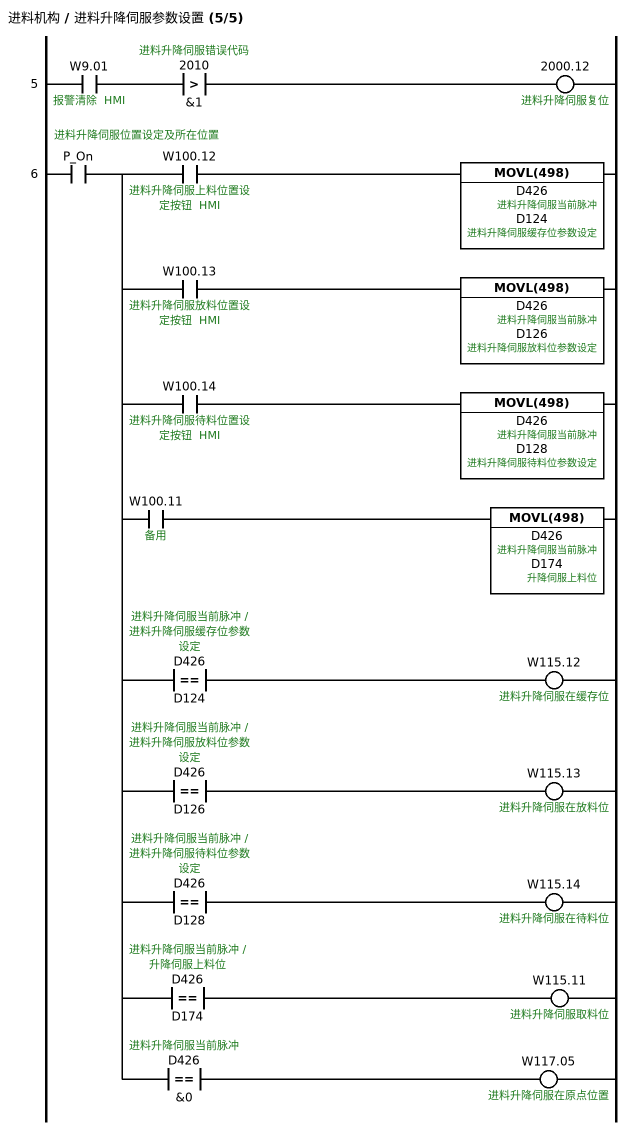
; [picture p144: 进料机构 / 进料升降伺服参数设置, rungs 5-6]
; rung 5
LD W9.01  ; 报警清除  HMI
AND>(320) 2010 &1  ; 进料升降伺服错误代码
OUT 2000.12  ; 进料升降伺服复位
; rung 6: 进料升降伺服位置设定及所在位置
LD P_On
OUT TR0
AND W100.12  ; 进料升降伺服上料位置设定按钮  HMI
MOVL(498) D426 D124  ; 进料升降伺服当前脉冲, 进料升降伺服缓存位参数设定
LD TR0
AND W100.13  ; 进料升降伺服放料位置设定按钮  HMI
MOVL(498) D426 D126  ; 进料升降伺服当前脉冲, 进料升降伺服放料位参数设定
LD TR0
AND W100.14  ; 进料升降伺服待料位置设定按钮  HMI
MOVL(498) D426 D128  ; 进料升降伺服当前脉冲, 进料升降伺服待料位参数设定
LD TR0
AND W100.11  ; 备用
MOVL(498) D426 D174  ; 进料升降伺服当前脉冲, 升降伺服上料位
LD TR0
AND=(300) D426 D124  ; 进料升降伺服当前脉冲, 进料升降伺服缓存位参数设定
OUT W115.12  ; 进料升降伺服在缓存位
LD TR0
AND=(300) D426 D126  ; 进料升降伺服当前脉冲, 进料升降伺服放料位参数设定
OUT W115.13  ; 进料升降伺服在放料位
LD TR0
AND=(300) D426 D128  ; 进料升降伺服当前脉冲, 进料升降伺服待料位参数设定
OUT W115.14  ; 进料升降伺服在待料位
LD TR0
AND=(300) D426 D174  ; 进料升降伺服当前脉冲, 升降伺服上料位
OUT W115.11  ; 进料升降伺服取料位
LD TR0
AND=(300) D426 &0  ; 进料升降伺服当前脉冲
OUT W117.05  ; 进料升降伺服在原点位置

### Section 进料旋转伺服参数设置

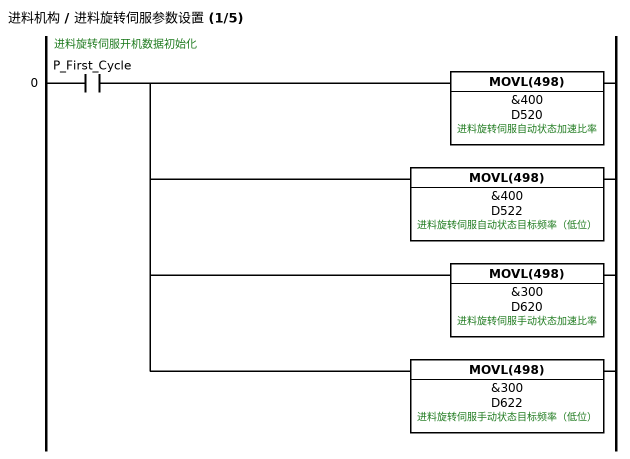
; rung 0: 进料旋转伺服开机数据初始化
LD P_First_Cycle
MOVL(498) &400 D520  ; 进料旋转伺服自动状态加速比率
MOVL(498) &400 D522  ; 进料旋转伺服自动状态目标频率（低位）
MOVL(498) &300 D620  ; 进料旋转伺服手动状态加速比率
MOVL(498) &300 D622  ; 进料旋转伺服手动状态目标频率（低位）

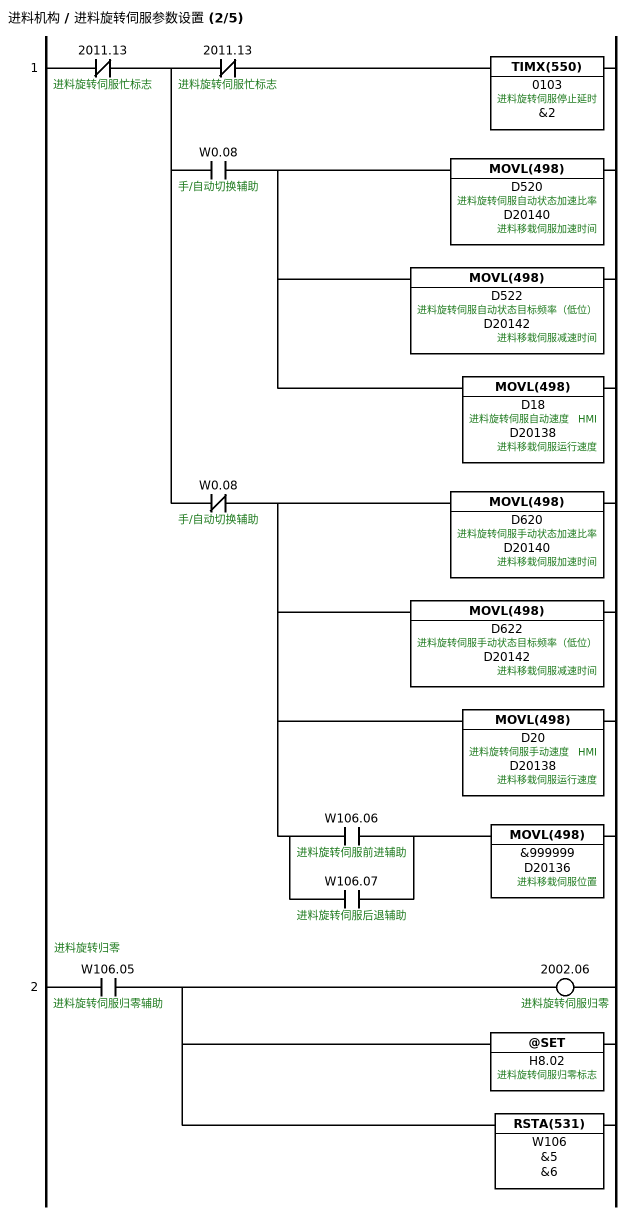
; rung 1
LDNOT 2011.13  ; 进料旋转伺服忙标志
OUT TR0
ANDNOT 2011.13  ; 进料旋转伺服忙标志
TIMX(550) 0103 &2  ; 进料旋转伺服停止延时
LD TR0
AND W0.08  ; 手/自动切换辅助
MOVL(498) D520 D20140  ; 进料旋转伺服自动状态加速比率, 进料移栽伺服加速时间
MOVL(498) D522 D20142  ; 进料旋转伺服自动状态目标频率（低位）, 进料移栽伺服减速时间
MOVL(498) D18 D20138  ; 进料旋转伺服自动速度   HMI, 进料移栽伺服运行速度
LD TR0
ANDNOT W0.08  ; 手/自动切换辅助
MOVL(498) D620 D20140  ; 进料旋转伺服手动状态加速比率, 进料移栽伺服加速时间
MOVL(498) D622 D20142  ; 进料旋转伺服手动状态目标频率（低位）, 进料移栽伺服减速时间
MOVL(498) D20 D20138  ; 进料旋转伺服手动速度   HMI, 进料移栽伺服运行速度
LD W106.06  ; 进料旋转伺服前进辅助
OR W106.07  ; 进料旋转伺服后退辅助
ANDLD
MOVL(498) &999999 D20136  ; 进料移栽伺服位置
; rung 2: 进料旋转归零
LD W106.05  ; 进料旋转伺服归零辅助
OUT 2002.06  ; 进料旋转伺服归零
@SET H8.02  ; 进料旋转伺服归零标志
RSTA(531) W106 &5 &6

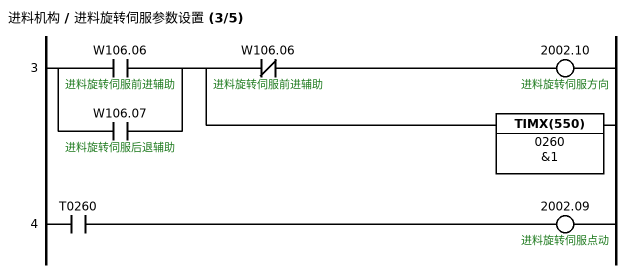
; rung 3
LD W106.06  ; 进料旋转伺服前进辅助
OR W106.07  ; 进料旋转伺服后退辅助
OUT TR0
ANDNOT W106.06  ; 进料旋转伺服前进辅助
OUT 2002.10  ; 进料旋转伺服方向
LD TR0
TIMX(550) 0260 &1
; rung 4
LD T0260
OUT 2002.09  ; 进料旋转伺服点动

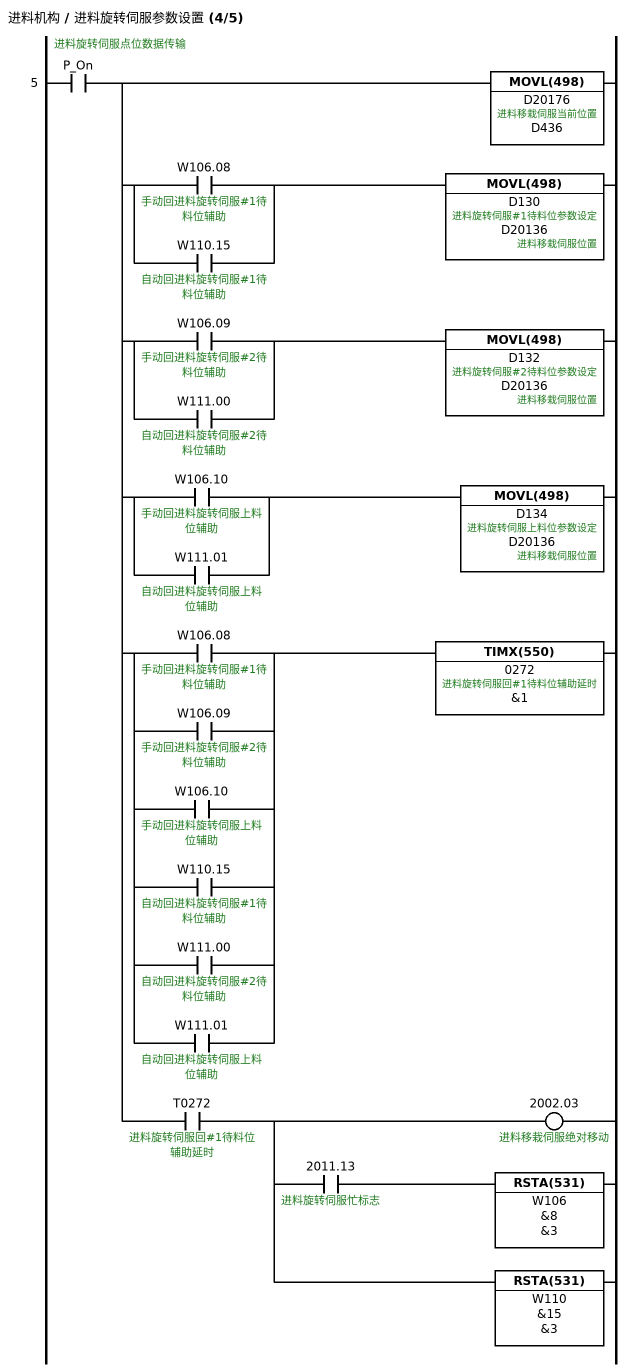
; rung 5: 进料旋转伺服点位数据传输
LD P_On
OUT TR0
MOVL(498) D20176 D436  ; 进料移栽伺服当前位置
LD W106.08  ; 手动回进料旋转伺服#1待料位辅助
OR W110.15  ; 自动回进料旋转伺服#1待料位辅助
ANDLD
MOVL(498) D130 D20136  ; 进料旋转伺服#1待料位参数设定, 进料移栽伺服位置
LD TR0
LD W106.09  ; 手动回进料旋转伺服#2待料位辅助
OR W111.00  ; 自动回进料旋转伺服#2待料位辅助
ANDLD
MOVL(498) D132 D20136  ; 进料旋转伺服#2待料位参数设定, 进料移栽伺服位置
LD TR0
LD W106.10  ; 手动回进料旋转伺服上料位辅助
OR W111.01  ; 自动回进料旋转伺服上料位辅助
ANDLD
MOVL(498) D134 D20136  ; 进料旋转伺服上料位参数设定, 进料移栽伺服位置
LD TR0
LD W106.08  ; 手动回进料旋转伺服#1待料位辅助
OR W106.09  ; 手动回进料旋转伺服#2待料位辅助
OR W106.10  ; 手动回进料旋转伺服上料位辅助
OR W110.15  ; 自动回进料旋转伺服#1待料位辅助
OR W111.00  ; 自动回进料旋转伺服#2待料位辅助
OR W111.01  ; 自动回进料旋转伺服上料位辅助
ANDLD
TIMX(550) 0272 &1  ; 进料旋转伺服回#1待料位辅助延时
LD TR0
AND T0272  ; 进料旋转伺服回#1待料位辅助延时
OUT TR0
OUT 2002.03  ; 进料移栽伺服绝对移动
AND 2011.13  ; 进料旋转伺服忙标志
RSTA(531) W106 &8 &3
LD TR0
RSTA(531) W110 &15 &3

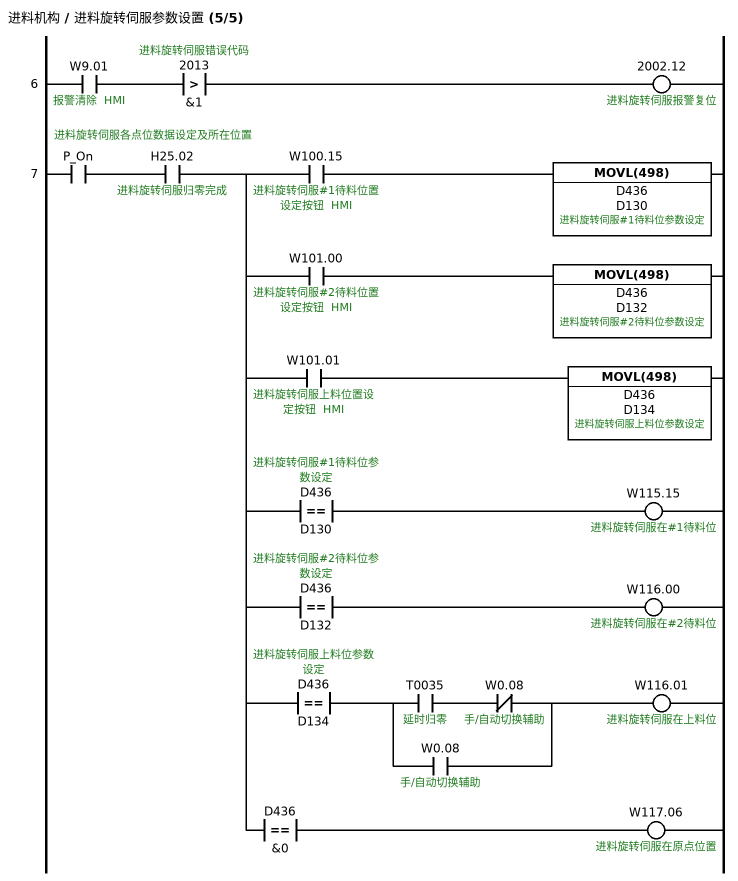
; rung 6
LD W9.01  ; 报警清除  HMI
AND>(320) 2013 &1  ; 进料旋转伺服错误代码
OUT 2002.12  ; 进料旋转伺服报警复位
; rung 7: 进料旋转伺服各点位数据设定及所在位置
LD P_On
AND H25.02  ; 进料旋转伺服归零完成
OUT TR0
AND W100.15  ; 进料旋转伺服#1待料位置设定按钮  HMI
MOVL(498) D436 D130  ; 进料旋转伺服#1待料位参数设定
LD TR0
AND W101.00  ; 进料旋转伺服#2待料位置设定按钮  HMI
MOVL(498) D436 D132  ; 进料旋转伺服#2待料位参数设定
LD TR0
AND W101.01  ; 进料旋转伺服上料位置设定按钮  HMI
MOVL(498) D436 D134  ; 进料旋转伺服上料位参数设定
LD TR0
AND=(300) D436 D130  ; 进料旋转伺服#1待料位参数设定
OUT W115.15  ; 进料旋转伺服在#1待料位
LD TR0
AND=(300) D436 D132  ; 进料旋转伺服#2待料位参数设定
OUT W116.00  ; 进料旋转伺服在#2待料位
LD TR0
AND=(300) D436 D134  ; 进料旋转伺服上料位参数设定
LD T0035  ; 延时归零
ANDNOT W0.08  ; 手/自动切换辅助
OR W0.08  ; 手/自动切换辅助
ANDLD
OUT W116.01  ; 进料旋转伺服在上料位
LD TR0
AND=(300) D436 &0
OUT W117.06  ; 进料旋转伺服在原点位置

### Section 扫码触发

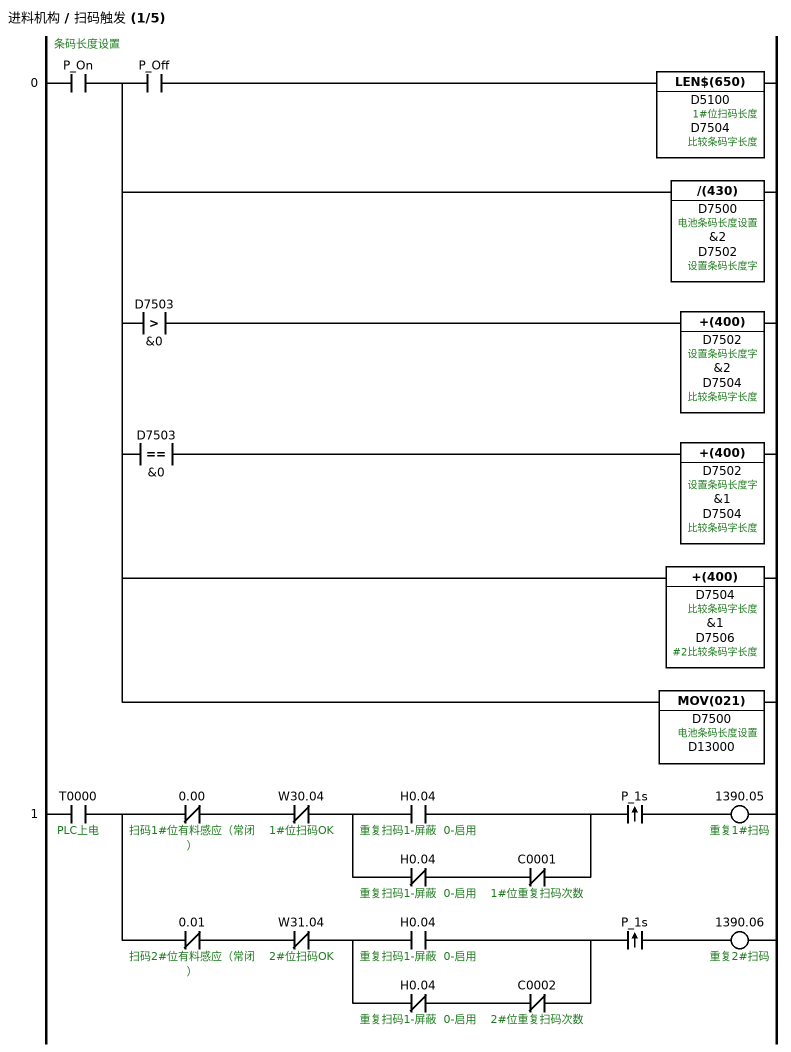
; rung 0: 条码长度设置
LD P_On
OUT TR0
AND P_Off
LEN$(650) D5100 D7504  ; 1#位扫码长度, 比较条码字长度
LD TR0
/(430) D7500 &2 D7502  ; 电池条码长度设置, 设置条码长度字
AND>(320) D7503 &0
+(400) D7502 &2 D7504  ; 设置条码长度字, 比较条码字长度
LD TR0
AND=(300) D7503 &0
+(400) D7502 &1 D7504  ; 设置条码长度字, 比较条码字长度
LD TR0
+(400) D7504 &1 D7506  ; 比较条码字长度, #2比较条码字长度
MOV(021) D7500 D13000  ; 电池条码长度设置
; rung 1
LD T0000  ; PLC上电
OUT TR0
ANDNOT 0.00  ; 扫码1#位有料感应（常闭）
ANDNOT W30.04  ; 1#位扫码OK
LD H0.04  ; 重复扫码1-屏蔽  0-启用
LDNOT H0.04  ; 重复扫码1-屏蔽  0-启用
ANDNOT C0001  ; 1#位重复扫码次数
ORLD
ANDLD
@AND P_1s
OUT 1390.05  ; 重复1#扫码
LD TR0
ANDNOT 0.01  ; 扫码2#位有料感应（常闭）
ANDNOT W31.04  ; 2#位扫码OK
LD H0.04  ; 重复扫码1-屏蔽  0-启用
LDNOT H0.04  ; 重复扫码1-屏蔽  0-启用
ANDNOT C0002  ; 2#位重复扫码次数
ORLD
ANDLD
@AND P_1s
OUT 1390.06  ; 重复2#扫码

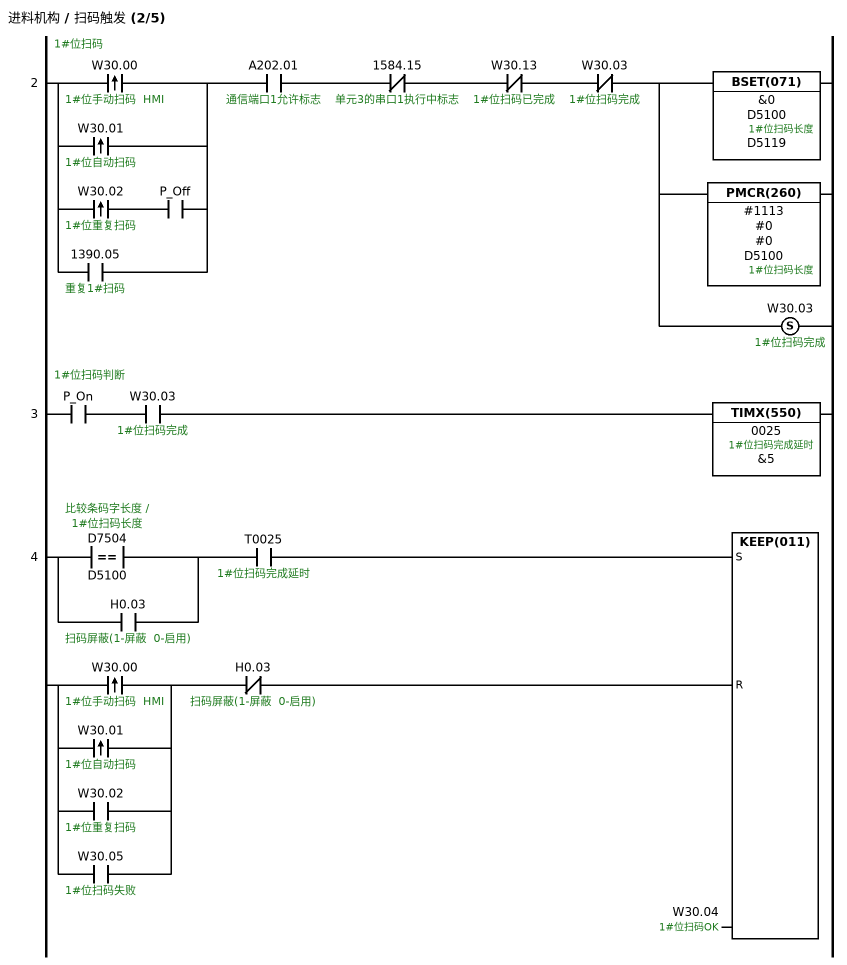
; rung 2: 1#位扫码
@LD W30.00  ; 1#位手动扫码  HMI
@OR W30.01  ; 1#位自动扫码
@LD W30.02  ; 1#位重复扫码
AND P_Off
ORLD
OR 1390.05  ; 重复1#扫码
AND A202.01  ; 通信端口1允许标志
ANDNOT 1584.15  ; 单元3的串口1执行中标志
ANDNOT W30.13  ; 1#位扫码已完成
ANDNOT W30.03  ; 1#位扫码完成
BSET(071) &0 D5100 D5119  ; 1#位扫码长度
PMCR(260) #1113 #0 #0 D5100  ; 1#位扫码长度
SET W30.03  ; 1#位扫码完成
; rung 3: 1#位扫码判断
LD P_On
AND W30.03  ; 1#位扫码完成
TIMX(550) 0025 &5  ; 1#位扫码完成延时
; rung 4
LD=(300) D7504 D5100  ; 比较条码字长度, 1#位扫码长度
OR H0.03  ; 扫码屏蔽(1-屏蔽  0-启用)
AND T0025  ; 1#位扫码完成延时
@LD W30.00  ; 1#位手动扫码  HMI
@OR W30.01  ; 1#位自动扫码
OR W30.02  ; 1#位重复扫码
OR W30.05  ; 1#位扫码失败
ANDNOT H0.03  ; 扫码屏蔽(1-屏蔽  0-启用)
KEEP(011) W30.04  ; 1#位扫码OK

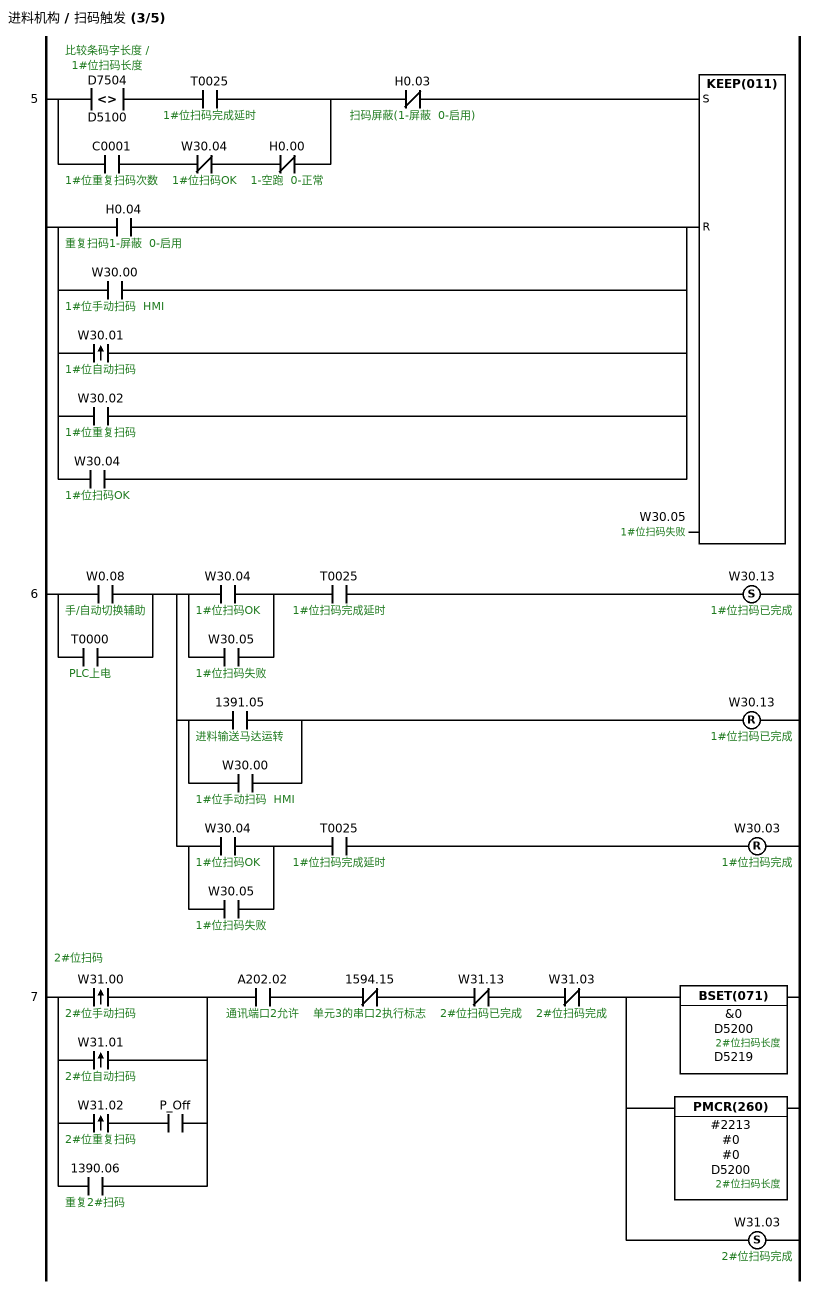
; rung 5
LD<>(305) D7504 D5100  ; 比较条码字长度, 1#位扫码长度
AND T0025  ; 1#位扫码完成延时
LD C0001  ; 1#位重复扫码次数
ANDNOT W30.04  ; 1#位扫码OK
ANDNOT H0.00  ; 1-空跑  0-正常
ORLD
ANDNOT H0.03  ; 扫码屏蔽(1-屏蔽  0-启用)
LD H0.04  ; 重复扫码1-屏蔽  0-启用
OR W30.00  ; 1#位手动扫码  HMI
@OR W30.01  ; 1#位自动扫码
OR W30.02  ; 1#位重复扫码
OR W30.04  ; 1#位扫码OK
KEEP(011) W30.05  ; 1#位扫码失败
; rung 6
LD W0.08  ; 手/自动切换辅助
OR T0000  ; PLC上电
OUT TR0
LD W30.04  ; 1#位扫码OK
OR W30.05  ; 1#位扫码失败
ANDLD
AND T0025  ; 1#位扫码完成延时
SET W30.13  ; 1#位扫码已完成
LD TR0
LD 1391.05  ; 进料输送马达运转
OR W30.00  ; 1#位手动扫码  HMI
ANDLD
RSET W30.13  ; 1#位扫码已完成
LD TR0
LD W30.04  ; 1#位扫码OK
OR W30.05  ; 1#位扫码失败
ANDLD
AND T0025  ; 1#位扫码完成延时
RSET W30.03  ; 1#位扫码完成
; rung 7: 2#位扫码
@LD W31.00  ; 2#位手动扫码
@OR W31.01  ; 2#位自动扫码
@LD W31.02  ; 2#位重复扫码
AND P_Off
ORLD
OR 1390.06  ; 重复2#扫码
AND A202.02  ; 通讯端口2允许
ANDNOT 1594.15  ; 单元3的串口2执行标志
ANDNOT W31.13  ; 2#位扫码已完成
ANDNOT W31.03  ; 2#位扫码完成
BSET(071) &0 D5200 D5219  ; 2#位扫码长度
PMCR(260) #2213 #0 #0 D5200  ; 2#位扫码长度
SET W31.03  ; 2#位扫码完成

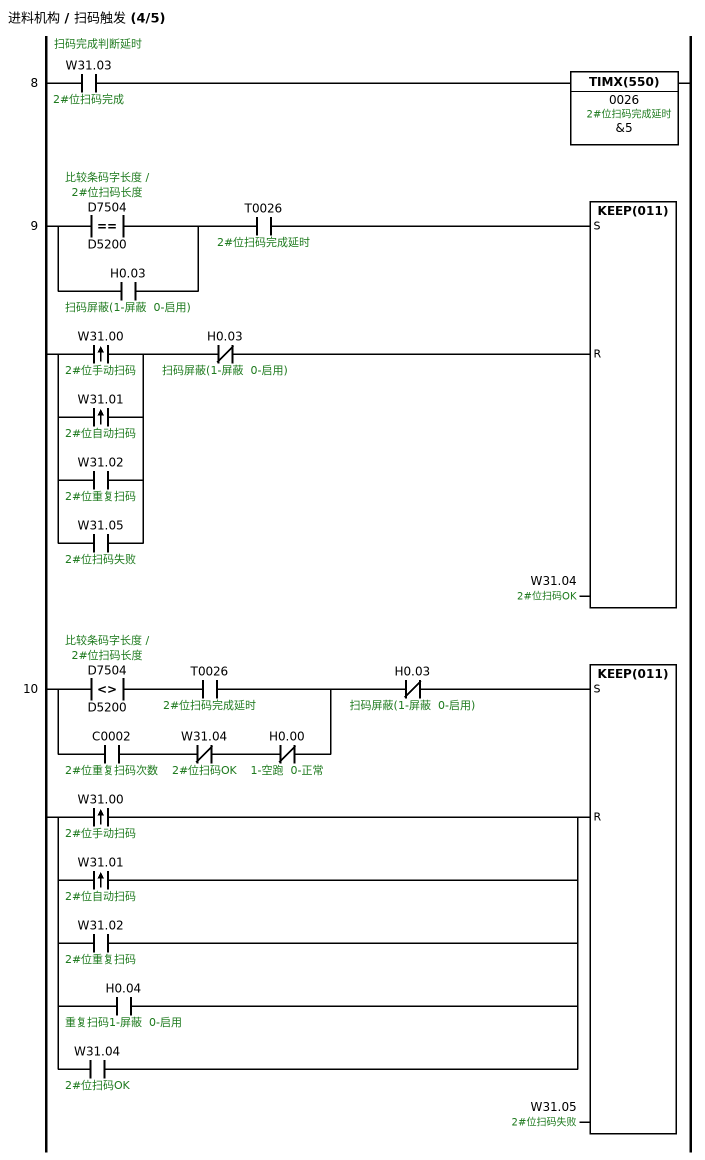
; rung 8: 扫码完成判断延时
LD W31.03  ; 2#位扫码完成
TIMX(550) 0026 &5  ; 2#位扫码完成延时
; rung 9
LD=(300) D7504 D5200  ; 比较条码字长度, 2#位扫码长度
OR H0.03  ; 扫码屏蔽(1-屏蔽  0-启用)
AND T0026  ; 2#位扫码完成延时
@LD W31.00  ; 2#位手动扫码
@OR W31.01  ; 2#位自动扫码
OR W31.02  ; 2#位重复扫码
OR W31.05  ; 2#位扫码失败
ANDNOT H0.03  ; 扫码屏蔽(1-屏蔽  0-启用)
KEEP(011) W31.04  ; 2#位扫码OK
; rung 10
LD<>(305) D7504 D5200  ; 比较条码字长度, 2#位扫码长度
AND T0026  ; 2#位扫码完成延时
LD C0002  ; 2#位重复扫码次数
ANDNOT W31.04  ; 2#位扫码OK
ANDNOT H0.00  ; 1-空跑  0-正常
ORLD
ANDNOT H0.03  ; 扫码屏蔽(1-屏蔽  0-启用)
@LD W31.00  ; 2#位手动扫码
@OR W31.01  ; 2#位自动扫码
OR W31.02  ; 2#位重复扫码
OR H0.04  ; 重复扫码1-屏蔽  0-启用
OR W31.04  ; 2#位扫码OK
KEEP(011) W31.05  ; 2#位扫码失败

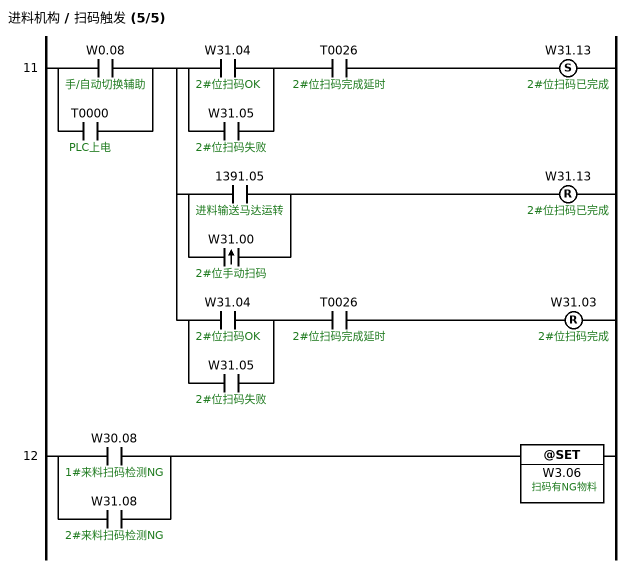
; rung 11
LD W0.08  ; 手/自动切换辅助
OR T0000  ; PLC上电
OUT TR0
LD W31.04  ; 2#位扫码OK
OR W31.05  ; 2#位扫码失败
ANDLD
AND T0026  ; 2#位扫码完成延时
SET W31.13  ; 2#位扫码已完成
LD TR0
LD 1391.05  ; 进料输送马达运转
@OR W31.00  ; 2#位手动扫码
ANDLD
RSET W31.13  ; 2#位扫码已完成
LD TR0
LD W31.04  ; 2#位扫码OK
OR W31.05  ; 2#位扫码失败
ANDLD
AND T0026  ; 2#位扫码完成延时
RSET W31.03  ; 2#位扫码完成
; rung 12
LD W30.08  ; 1#来料扫码检测NG
OR W31.08  ; 2#来料扫码检测NG
@SET W3.06  ; 扫码有NG物料

### Section 进料机构输出

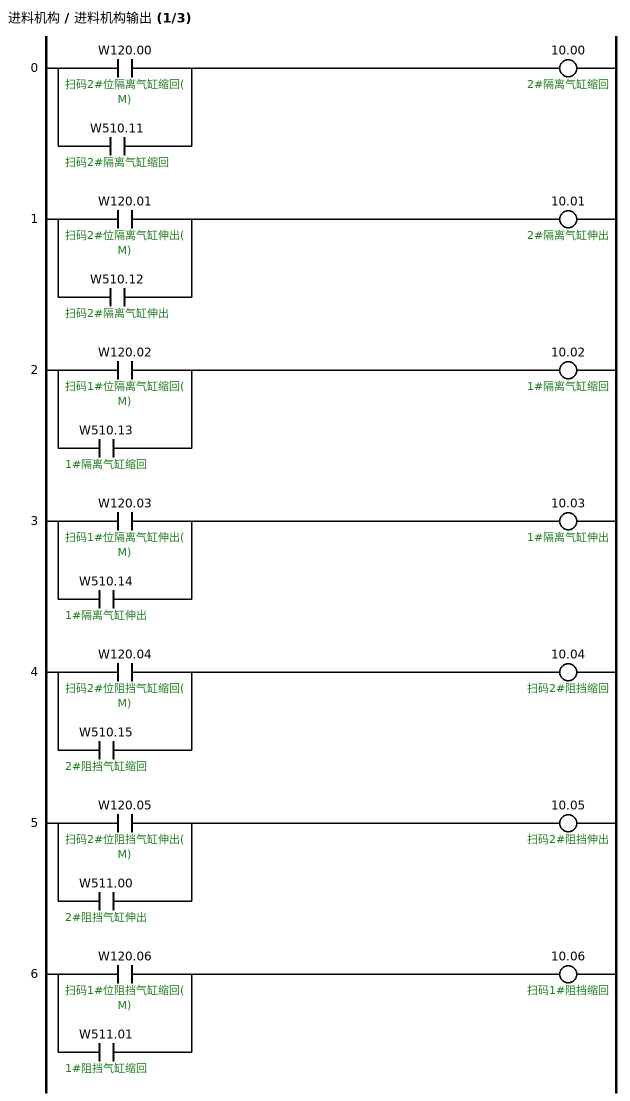
; rung 0
LD W120.00  ; 扫码2#位隔离气缸缩回(M)
OR W510.11  ; 扫码2#隔离气缸缩回
OUT 10.00  ; 2#隔离气缸缩回
; rung 1
LD W120.01  ; 扫码2#位隔离气缸伸出(M)
OR W510.12  ; 扫码2#隔离气缸伸出
OUT 10.01  ; 2#隔离气缸伸出
; rung 2
LD W120.02  ; 扫码1#位隔离气缸缩回(M)
OR W510.13  ; 1#隔离气缸缩回
OUT 10.02  ; 1#隔离气缸缩回
; rung 3
LD W120.03  ; 扫码1#位隔离气缸伸出(M)
OR W510.14  ; 1#隔离气缸伸出
OUT 10.03  ; 1#隔离气缸伸出
; rung 4
LD W120.04  ; 扫码2#位阻挡气缸缩回(M)
OR W510.15  ; 2#阻挡气缸缩回
OUT 10.04  ; 扫码2#阻挡缩回
; rung 5
LD W120.05  ; 扫码2#位阻挡气缸伸出(M)
OR W511.00  ; 2#阻挡气缸伸出
OUT 10.05  ; 扫码2#阻挡伸出
; rung 6
LD W120.06  ; 扫码1#位阻挡气缸缩回(M)
OR W511.01  ; 1#阻挡气缸缩回
OUT 10.06  ; 扫码1#阻挡缩回

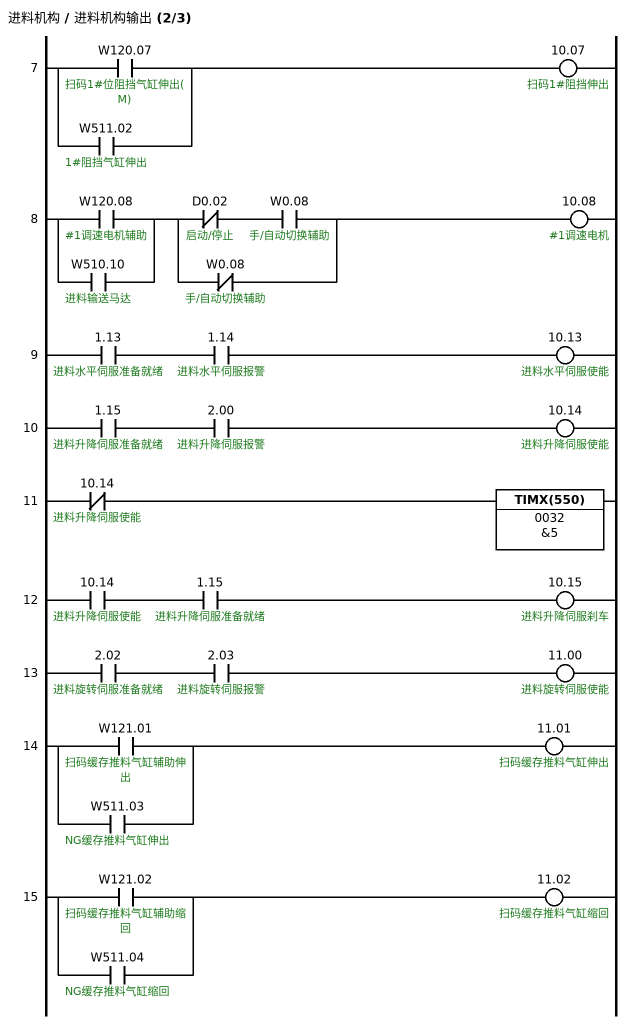
; rung 7
LD W120.07  ; 扫码1#位阻挡气缸伸出(M)
OR W511.02  ; 1#阻挡气缸伸出
OUT 10.07  ; 扫码1#阻挡伸出
; rung 8
LD W120.08  ; #1调速电机辅助
OR W510.10  ; 进料输送马达
LDNOT D0.02  ; 启动/停止
AND W0.08  ; 手/自动切换辅助
ORNOT W0.08  ; 手/自动切换辅助
ANDLD
OUT 10.08  ; #1调速电机
; rung 9
LD 1.13  ; 进料水平伺服准备就绪
AND 1.14  ; 进料水平伺服报警
OUT 10.13  ; 进料水平伺服使能
; rung 10
LD 1.15  ; 进料升降伺服准备就绪
AND 2.00  ; 进料升降伺服报警
OUT 10.14  ; 进料升降伺服使能
; rung 11
LDNOT 10.14  ; 进料升降伺服使能
TIMX(550) 0032 &5
; rung 12
LD 10.14  ; 进料升降伺服使能
AND 1.15  ; 进料升降伺服准备就绪
OUT 10.15  ; 进料升降伺服刹车
; rung 13
LD 2.02  ; 进料旋转伺服准备就绪
AND 2.03  ; 进料旋转伺服报警
OUT 11.00  ; 进料旋转伺服使能
; rung 14
LD W121.01  ; 扫码缓存推料气缸辅助伸出
OR W511.03  ; NG缓存推料气缸伸出
OUT 11.01  ; 扫码缓存推料气缸伸出
; rung 15
LD W121.02  ; 扫码缓存推料气缸辅助缩回
OR W511.04  ; NG缓存推料气缸缩回
OUT 11.02  ; 扫码缓存推料气缸缩回

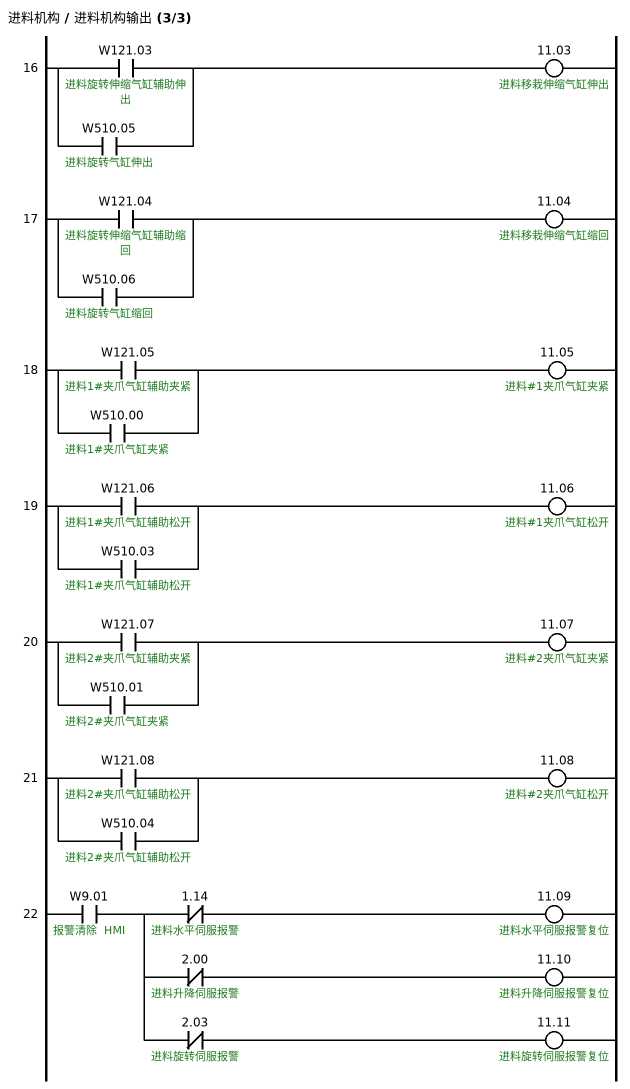
; rung 16
LD W121.03  ; 进料旋转伸缩气缸辅助伸出
OR W510.05  ; 进料旋转气缸伸出
OUT 11.03  ; 进料移栽伸缩气缸伸出
; rung 17
LD W121.04  ; 进料旋转伸缩气缸辅助缩回
OR W510.06  ; 进料旋转气缸缩回
OUT 11.04  ; 进料移栽伸缩气缸缩回
; rung 18
LD W121.05  ; 进料1#夹爪气缸辅助夹紧
OR W510.00  ; 进料1#夹爪气缸夹紧
OUT 11.05  ; 进料#1夹爪气缸夹紧
; rung 19
LD W121.06  ; 进料1#夹爪气缸辅助松开
OR W510.03  ; 进料1#夹爪气缸辅助松开
OUT 11.06  ; 进料#1夹爪气缸松开
; rung 20
LD W121.07  ; 进料2#夹爪气缸辅助夹紧
OR W510.01  ; 进料2#夹爪气缸夹紧
OUT 11.07  ; 进料#2夹爪气缸夹紧
; rung 21
LD W121.08  ; 进料2#夹爪气缸辅助松开
OR W510.04  ; 进料2#夹爪气缸辅助松开
OUT 11.08  ; 进料#2夹爪气缸松开
; rung 22
LD W9.01  ; 报警清除  HMI
OUT TR0
ANDNOT 1.14  ; 进料水平伺服报警
OUT 11.09  ; 进料水平伺服报警复位
LD TR0
ANDNOT 2.00  ; 进料升降伺服报警
OUT 11.10  ; 进料升降伺服报警复位
LD TR0
ANDNOT 2.03  ; 进料旋转伺服报警
OUT 11.11  ; 进料旋转伺服报警复位

### Section 工站复位

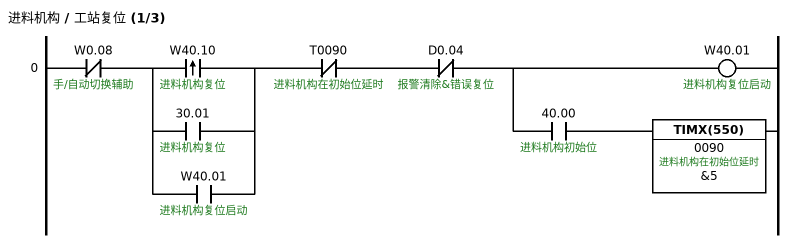
; rung 0
LDNOT W0.08  ; 手/自动切换辅助
@LD W40.10  ; 进料机构复位
OR 30.01  ; 进料机构复位
OR W40.01  ; 进料机构复位启动
ANDLD
ANDNOT T0090  ; 进料机构在初始位延时
ANDNOT D0.04  ; 报警清除&错误复位
OUT W40.01  ; 进料机构复位启动
AND 40.00  ; 进料机构初始位
TIMX(550) 0090 &5  ; 进料机构在初始位延时

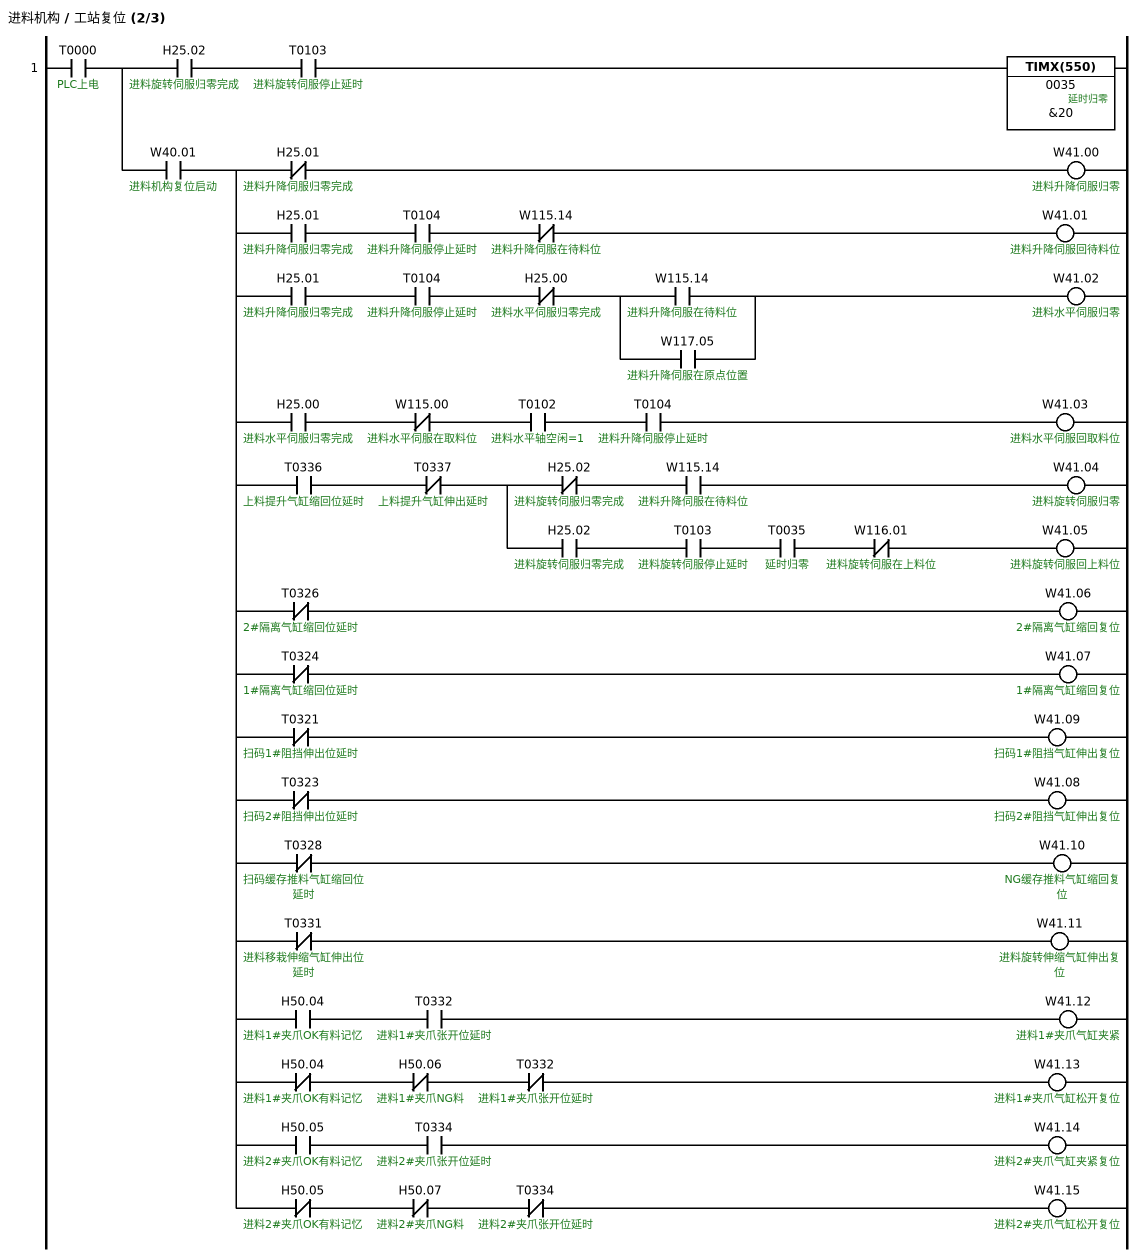
; rung 1
LD T0000  ; PLC上电
OUT TR0
AND H25.02  ; 进料旋转伺服归零完成
AND T0103  ; 进料旋转伺服停止延时
TIMX(550) 0035 &20  ; 延时归零
LD TR0
AND W40.01  ; 进料机构复位启动
OUT TR0
ANDNOT H25.01  ; 进料升降伺服归零完成
OUT W41.00  ; 进料升降伺服归零
LD TR0
AND H25.01  ; 进料升降伺服归零完成
AND T0104  ; 进料升降伺服停止延时
ANDNOT W115.14  ; 进料升降伺服在待料位
OUT W41.01  ; 进料升降伺服回待料位
LD TR0
AND H25.01  ; 进料升降伺服归零完成
AND T0104  ; 进料升降伺服停止延时
ANDNOT H25.00  ; 进料水平伺服归零完成
LD W115.14  ; 进料升降伺服在待料位
OR W117.05  ; 进料升降伺服在原点位置
ANDLD
OUT W41.02  ; 进料水平伺服归零
LD TR0
AND H25.00  ; 进料水平伺服归零完成
ANDNOT W115.00  ; 进料水平伺服在取料位
AND T0102  ; 进料水平轴空闲=1
AND T0104  ; 进料升降伺服停止延时
OUT W41.03  ; 进料水平伺服回取料位
LD TR0
AND T0336  ; 上料提升气缸缩回位延时
ANDNOT T0337  ; 上料提升气缸伸出延时
OUT TR1
ANDNOT H25.02  ; 进料旋转伺服归零完成
AND W115.14  ; 进料升降伺服在待料位
OUT W41.04  ; 进料旋转伺服归零
LD TR1
AND H25.02  ; 进料旋转伺服归零完成
AND T0103  ; 进料旋转伺服停止延时
AND T0035  ; 延时归零
ANDNOT W116.01  ; 进料旋转伺服在上料位
OUT W41.05  ; 进料旋转伺服回上料位
LD TR0
ANDNOT T0326  ; 2#隔离气缸缩回位延时
OUT W41.06  ; 2#隔离气缸缩回复位
LD TR0
ANDNOT T0324  ; 1#隔离气缸缩回位延时
OUT W41.07  ; 1#隔离气缸缩回复位
LD TR0
ANDNOT T0321  ; 扫码1#阻挡伸出位延时
OUT W41.09  ; 扫码1#阻挡气缸伸出复位
LD TR0
ANDNOT T0323  ; 扫码2#阻挡伸出位延时
OUT W41.08  ; 扫码2#阻挡气缸伸出复位
LD TR0
ANDNOT T0328  ; 扫码缓存推料气缸缩回位延时
OUT W41.10  ; NG缓存推料气缸缩回复位
LD TR0
ANDNOT T0331  ; 进料移栽伸缩气缸伸出位延时
OUT W41.11  ; 进料旋转伸缩气缸伸出复位
LD TR0
AND H50.04  ; 进料1#夹爪OK有料记忆
AND T0332  ; 进料1#夹爪张开位延时
OUT W41.12  ; 进料1#夹爪气缸夹紧
LD TR0
ANDNOT H50.04  ; 进料1#夹爪OK有料记忆
ANDNOT H50.06  ; 进料1#夹爪NG料
ANDNOT T0332  ; 进料1#夹爪张开位延时
OUT W41.13  ; 进料1#夹爪气缸松开复位
LD TR0
AND H50.05  ; 进料2#夹爪OK有料记忆
AND T0334  ; 进料2#夹爪张开位延时
OUT W41.14  ; 进料2#夹爪气缸夹紧复位
LD TR0
ANDNOT H50.05  ; 进料2#夹爪OK有料记忆
ANDNOT H50.07  ; 进料2#夹爪NG料
ANDNOT T0334  ; 进料2#夹爪张开位延时
OUT W41.15  ; 进料2#夹爪气缸松开复位

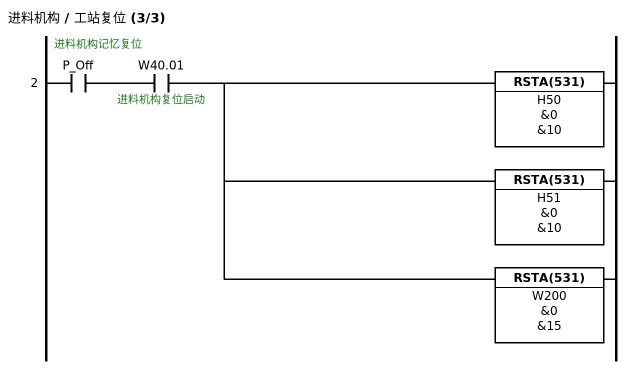
; rung 2: 进料机构记忆复位
LD P_Off
AND W40.01  ; 进料机构复位启动
RSTA(531) H50 &0 &10
RSTA(531) H51 &0 &10
RSTA(531) W200 &0 &15

### Section END
; rung 0
END(001)

## Program 上下料机构 (cyclic task 2)

### Section 上下料机构自动

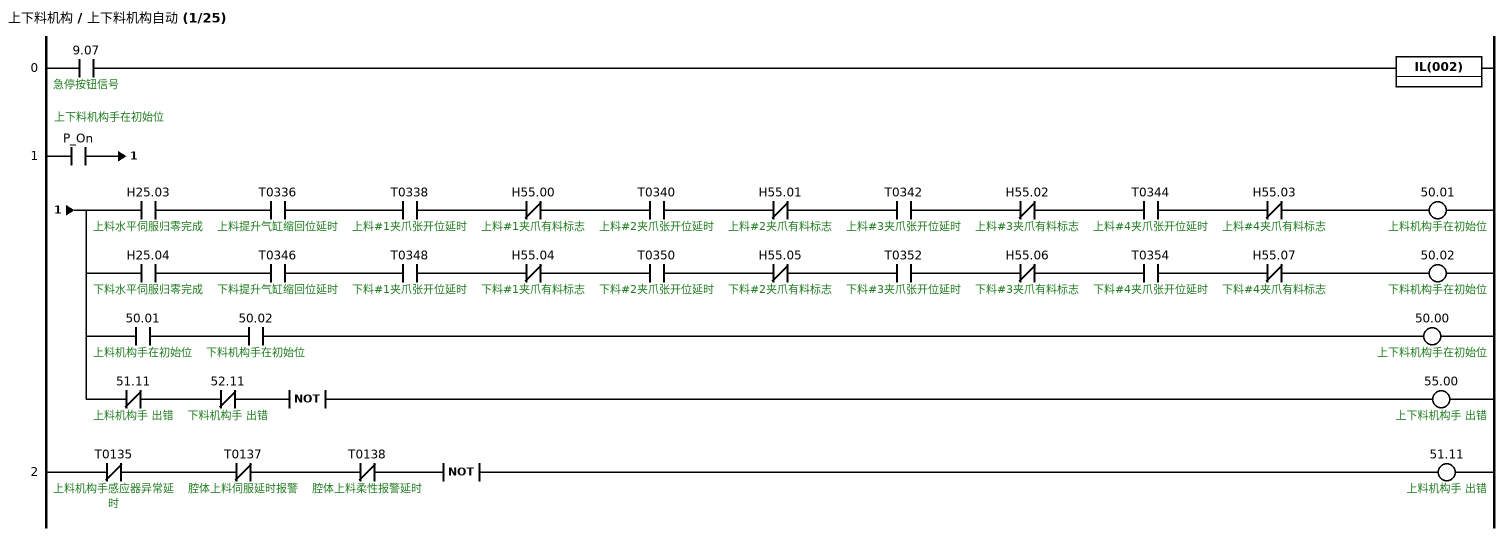
; rung 0
LD 9.07  ; 急停按钮信号
IL(002)
; rung 1: 上下料机构手在初始位
LD P_On
OUT TR0
AND H25.03  ; 上料水平伺服归零完成
AND T0336  ; 上料提升气缸缩回位延时
AND T0338  ; 上料#1夹爪张开位延时
ANDNOT H55.00  ; 上料#1夹爪有料标志
AND T0340  ; 上料#2夹爪张开位延时
ANDNOT H55.01  ; 上料#2夹爪有料标志
AND T0342  ; 上料#3夹爪张开位延时
ANDNOT H55.02  ; 上料#3夹爪有料标志
AND T0344  ; 上料#4夹爪张开位延时
ANDNOT H55.03  ; 上料#4夹爪有料标志
OUT 50.01  ; 上料机构手在初始位
LD TR0
AND H25.04  ; 下料水平伺服归零完成
AND T0346  ; 下料提升气缸缩回位延时
AND T0348  ; 下料#1夹爪张开位延时
ANDNOT H55.04  ; 下料#1夹爪有料标志
AND T0350  ; 下料#2夹爪张开位延时
ANDNOT H55.05  ; 下料#2夹爪有料标志
AND T0352  ; 下料#3夹爪张开位延时
ANDNOT H55.06  ; 下料#3夹爪有料标志
AND T0354  ; 下料#4夹爪张开位延时
ANDNOT H55.07  ; 下料#4夹爪有料标志
OUT 50.02  ; 下料机构手在初始位
LD TR0
AND 50.01  ; 上料机构手在初始位
AND 50.02  ; 下料机构手在初始位
OUT 50.00  ; 上下料机构手在初始位
LD TR0
ANDNOT 51.11  ; 上料机构手 出错
ANDNOT 52.11  ; 下料机构手 出错
NOT(520)
OUT 55.00  ; 上下料机构手 出错
; rung 2
LDNOT T0135  ; 上料机构手感应器异常延时
ANDNOT T0137  ; 腔体上料伺服延时报警
ANDNOT T0138  ; 腔体上料柔性报警延时
NOT(520)
OUT 51.11  ; 上料机构手 出错

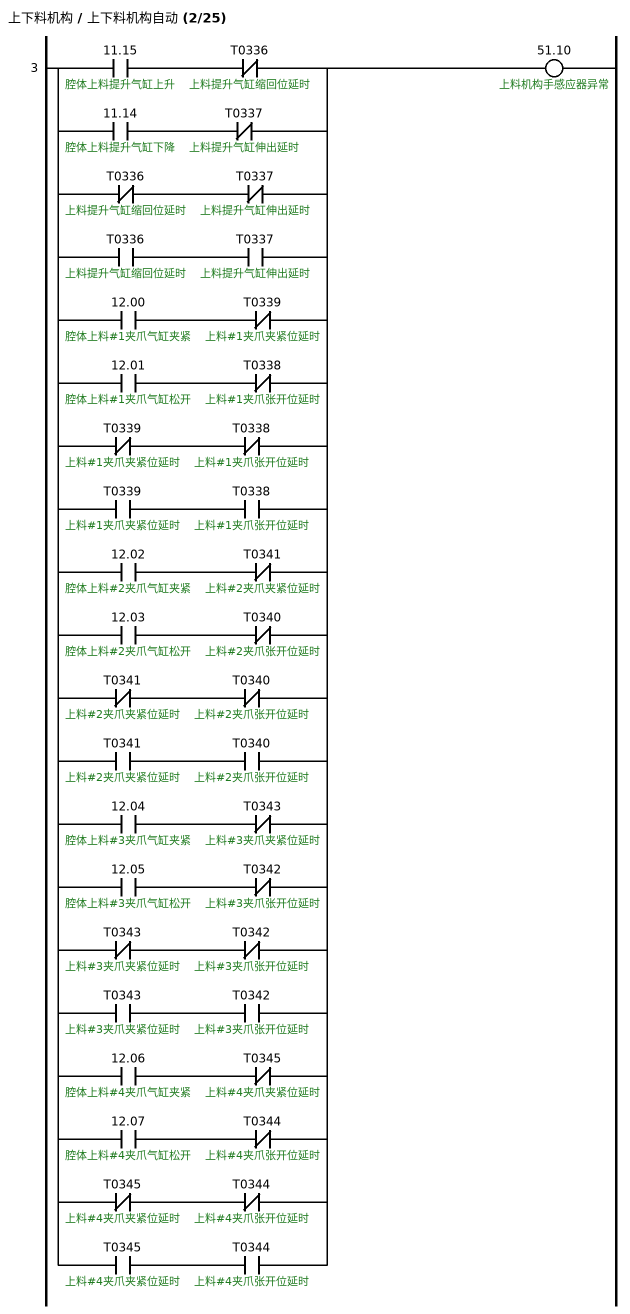
; rung 3
LD 11.15  ; 腔体上料提升气缸上升
ANDNOT T0336  ; 上料提升气缸缩回位延时
LD 11.14  ; 腔体上料提升气缸下降
ANDNOT T0337  ; 上料提升气缸伸出延时
ORLD
LDNOT T0336  ; 上料提升气缸缩回位延时
ANDNOT T0337  ; 上料提升气缸伸出延时
ORLD
LD T0336  ; 上料提升气缸缩回位延时
AND T0337  ; 上料提升气缸伸出延时
ORLD
LD 12.00  ; 腔体上料#1夹爪气缸夹紧
ANDNOT T0339  ; 上料#1夹爪夹紧位延时
ORLD
LD 12.01  ; 腔体上料#1夹爪气缸松开
ANDNOT T0338  ; 上料#1夹爪张开位延时
ORLD
LDNOT T0339  ; 上料#1夹爪夹紧位延时
ANDNOT T0338  ; 上料#1夹爪张开位延时
ORLD
LD T0339  ; 上料#1夹爪夹紧位延时
AND T0338  ; 上料#1夹爪张开位延时
ORLD
LD 12.02  ; 腔体上料#2夹爪气缸夹紧
ANDNOT T0341  ; 上料#2夹爪夹紧位延时
ORLD
LD 12.03  ; 腔体上料#2夹爪气缸松开
ANDNOT T0340  ; 上料#2夹爪张开位延时
ORLD
LDNOT T0341  ; 上料#2夹爪夹紧位延时
ANDNOT T0340  ; 上料#2夹爪张开位延时
ORLD
LD T0341  ; 上料#2夹爪夹紧位延时
AND T0340  ; 上料#2夹爪张开位延时
ORLD
LD 12.04  ; 腔体上料#3夹爪气缸夹紧
ANDNOT T0343  ; 上料#3夹爪夹紧位延时
ORLD
LD 12.05  ; 腔体上料#3夹爪气缸松开
ANDNOT T0342  ; 上料#3夹爪张开位延时
ORLD
LDNOT T0343  ; 上料#3夹爪夹紧位延时
ANDNOT T0342  ; 上料#3夹爪张开位延时
ORLD
LD T0343  ; 上料#3夹爪夹紧位延时
AND T0342  ; 上料#3夹爪张开位延时
ORLD
LD 12.06  ; 腔体上料#4夹爪气缸夹紧
ANDNOT T0345  ; 上料#4夹爪夹紧位延时
ORLD
LD 12.07  ; 腔体上料#4夹爪气缸松开
ANDNOT T0344  ; 上料#4夹爪张开位延时
ORLD
LDNOT T0345  ; 上料#4夹爪夹紧位延时
ANDNOT T0344  ; 上料#4夹爪张开位延时
ORLD
LD T0345  ; 上料#4夹爪夹紧位延时
AND T0344  ; 上料#4夹爪张开位延时
ORLD
OUT 51.10  ; 上料机构手感应器异常

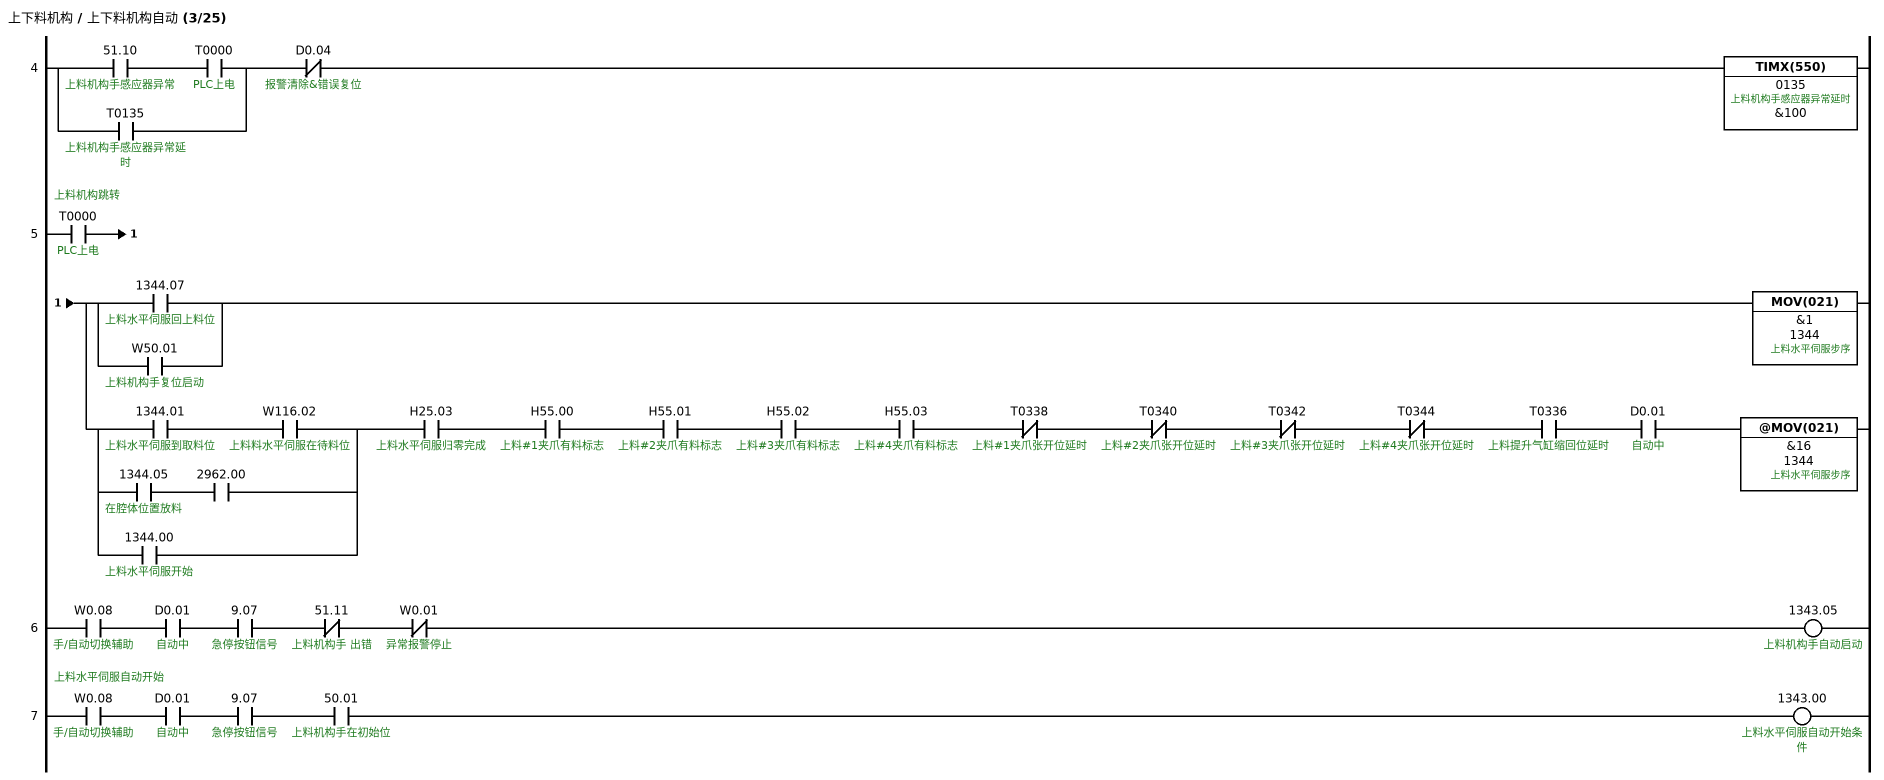
; rung 4
LD 51.10  ; 上料机构手感应器异常
AND T0000  ; PLC上电
OR T0135  ; 上料机构手感应器异常延时
ANDNOT D0.04  ; 报警清除&错误复位
TIMX(550) 0135 &100  ; 上料机构手感应器异常延时
; rung 5: 上料机构跳转
LD T0000  ; PLC上电
OUT TR0
LD 1344.07  ; 上料水平伺服回上料位
OR W50.01  ; 上料机构手复位启动
ANDLD
MOV(021) &1 1344  ; 上料水平伺服步序
LD TR0
LD 1344.01  ; 上料水平伺服到取料位
AND W116.02  ; 上料料水平伺服在待料位
LD 1344.05  ; 在腔体位置放料
AND 2962.00
ORLD
OR 1344.00  ; 上料水平伺服开始
ANDLD
AND H25.03  ; 上料水平伺服归零完成
AND H55.00  ; 上料#1夹爪有料标志
AND H55.01  ; 上料#2夹爪有料标志
AND H55.02  ; 上料#3夹爪有料标志
AND H55.03  ; 上料#4夹爪有料标志
ANDNOT T0338  ; 上料#1夹爪张开位延时
ANDNOT T0340  ; 上料#2夹爪张开位延时
ANDNOT T0342  ; 上料#3夹爪张开位延时
ANDNOT T0344  ; 上料#4夹爪张开位延时
AND T0336  ; 上料提升气缸缩回位延时
AND D0.01  ; 自动中
@MOV(021) &16 1344  ; 上料水平伺服步序
; rung 6
LD W0.08  ; 手/自动切换辅助
AND D0.01  ; 自动中
AND 9.07  ; 急停按钮信号
ANDNOT 51.11  ; 上料机构手 出错
ANDNOT W0.01  ; 异常报警停止
OUT 1343.05  ; 上料机构手自动启动
; rung 7: 上料水平伺服自动开始
LD W0.08  ; 手/自动切换辅助
AND D0.01  ; 自动中
AND 9.07  ; 急停按钮信号
AND 50.01  ; 上料机构手在初始位
OUT 1343.00  ; 上料水平伺服自动开始条件

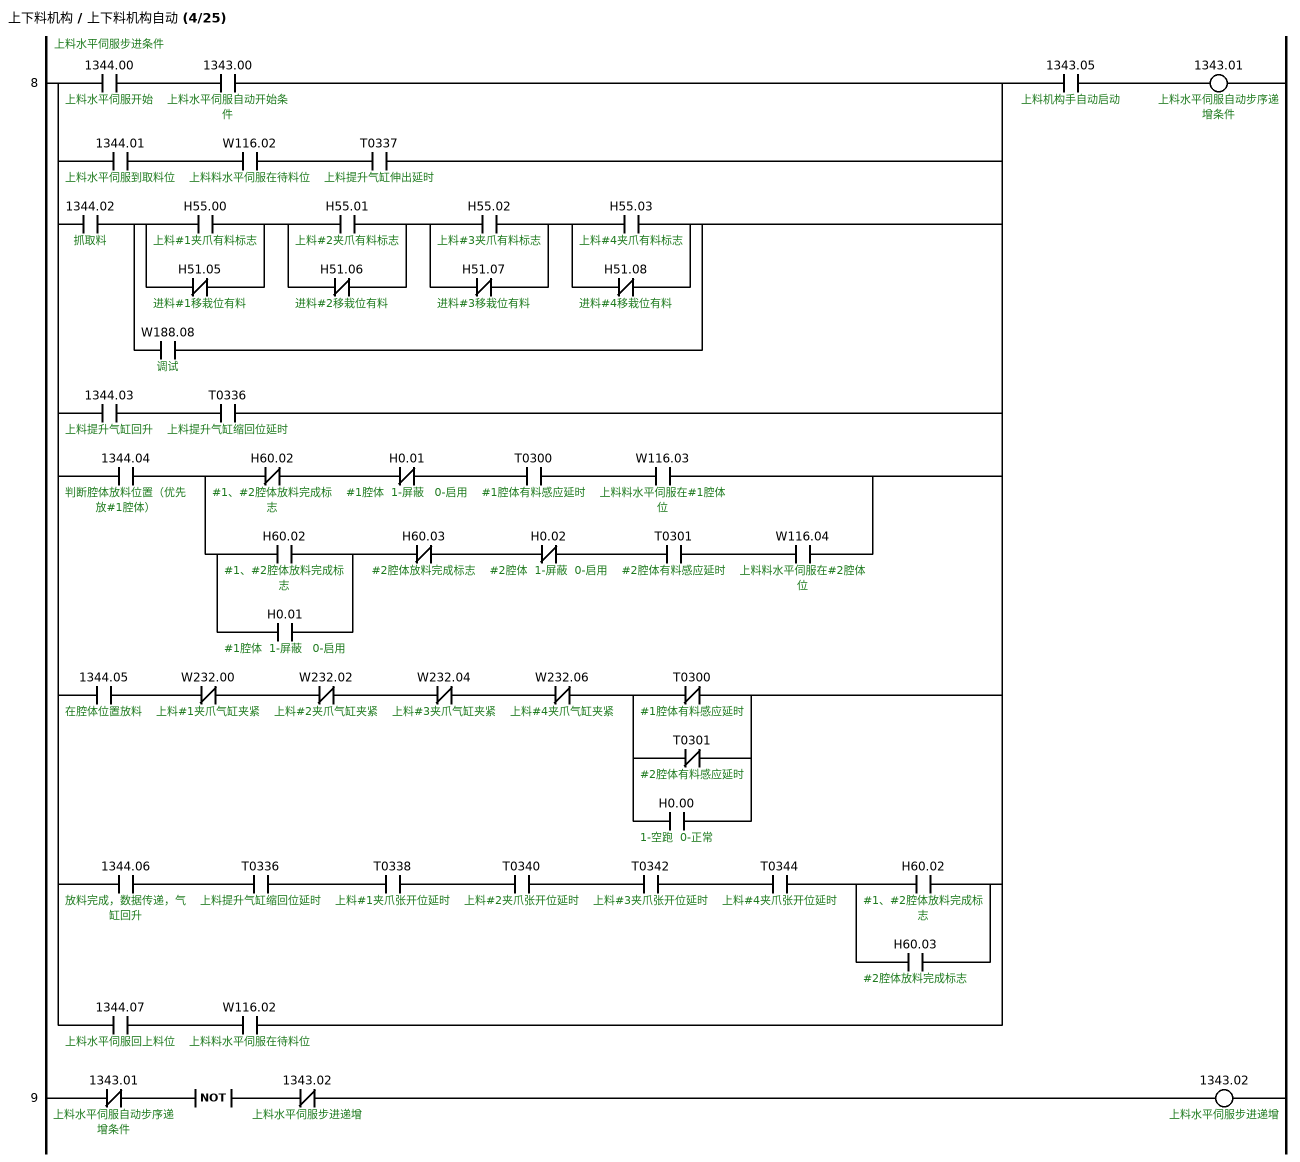
; rung 8: 上料水平伺服步进条件
LD 1344.00  ; 上料水平伺服开始
AND 1343.00  ; 上料水平伺服自动开始条件
LD 1344.01  ; 上料水平伺服到取料位
AND W116.02  ; 上料料水平伺服在待料位
AND T0337  ; 上料提升气缸伸出延时
ORLD
LD 1344.02  ; 抓取料
LD H55.00  ; 上料#1夹爪有料标志
ORNOT H51.05  ; 进料#1移栽位有料
LD H55.01  ; 上料#2夹爪有料标志
ORNOT H51.06  ; 进料#2移栽位有料
ANDLD
LD H55.02  ; 上料#3夹爪有料标志
ORNOT H51.07  ; 进料#3移栽位有料
ANDLD
LD H55.03  ; 上料#4夹爪有料标志
ORNOT H51.08  ; 进料#4移栽位有料
ANDLD
OR W188.08  ; 调试
ANDLD
ORLD
LD 1344.03  ; 上料提升气缸回升
AND T0336  ; 上料提升气缸缩回位延时
ORLD
LD 1344.04  ; 判断腔体放料位置（优先放#1腔体）
LDNOT H60.02  ; #1、#2腔体放料完成标志
ANDNOT H0.01  ; #1腔体  1-屏蔽   0-启用
AND T0300  ; #1腔体有料感应延时
AND W116.03  ; 上料料水平伺服在#1腔体位
LD H60.02  ; #1、#2腔体放料完成标志
OR H0.01  ; #1腔体  1-屏蔽   0-启用
ANDNOT H60.03  ; #2腔体放料完成标志
ANDNOT H0.02  ; #2腔体  1-屏蔽  0-启用
AND T0301  ; #2腔体有料感应延时
AND W116.04  ; 上料料水平伺服在#2腔体位
ORLD
ANDLD
ORLD
LD 1344.05  ; 在腔体位置放料
ANDNOT W232.00  ; 上料#1夹爪气缸夹紧
ANDNOT W232.02  ; 上料#2夹爪气缸夹紧
ANDNOT W232.04  ; 上料#3夹爪气缸夹紧
ANDNOT W232.06  ; 上料#4夹爪气缸夹紧
LDNOT T0300  ; #1腔体有料感应延时
ORNOT T0301  ; #2腔体有料感应延时
OR H0.00  ; 1-空跑  0-正常
ANDLD
ORLD
LD 1344.06  ; 放料完成，数据传递，气缸回升
AND T0336  ; 上料提升气缸缩回位延时
AND T0338  ; 上料#1夹爪张开位延时
AND T0340  ; 上料#2夹爪张开位延时
AND T0342  ; 上料#3夹爪张开位延时
AND T0344  ; 上料#4夹爪张开位延时
LD H60.02  ; #1、#2腔体放料完成标志
OR H60.03  ; #2腔体放料完成标志
ANDLD
ORLD
LD 1344.07  ; 上料水平伺服回上料位
AND W116.02  ; 上料料水平伺服在待料位
ORLD
AND 1343.05  ; 上料机构手自动启动
OUT 1343.01  ; 上料水平伺服自动步序递增条件
; rung 9
LDNOT 1343.01  ; 上料水平伺服自动步序递增条件
NOT(520)
ANDNOT 1343.02  ; 上料水平伺服步进递增
OUT 1343.02  ; 上料水平伺服步进递增

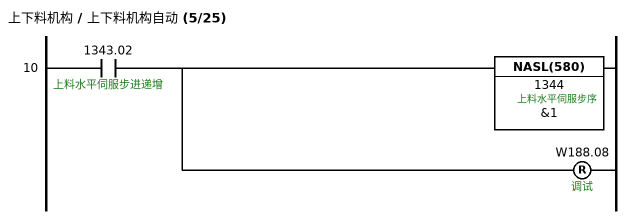
; rung 10
LD 1343.02  ; 上料水平伺服步进递增
NASL(580) 1344 &1  ; 上料水平伺服步序
RSET W188.08  ; 调试

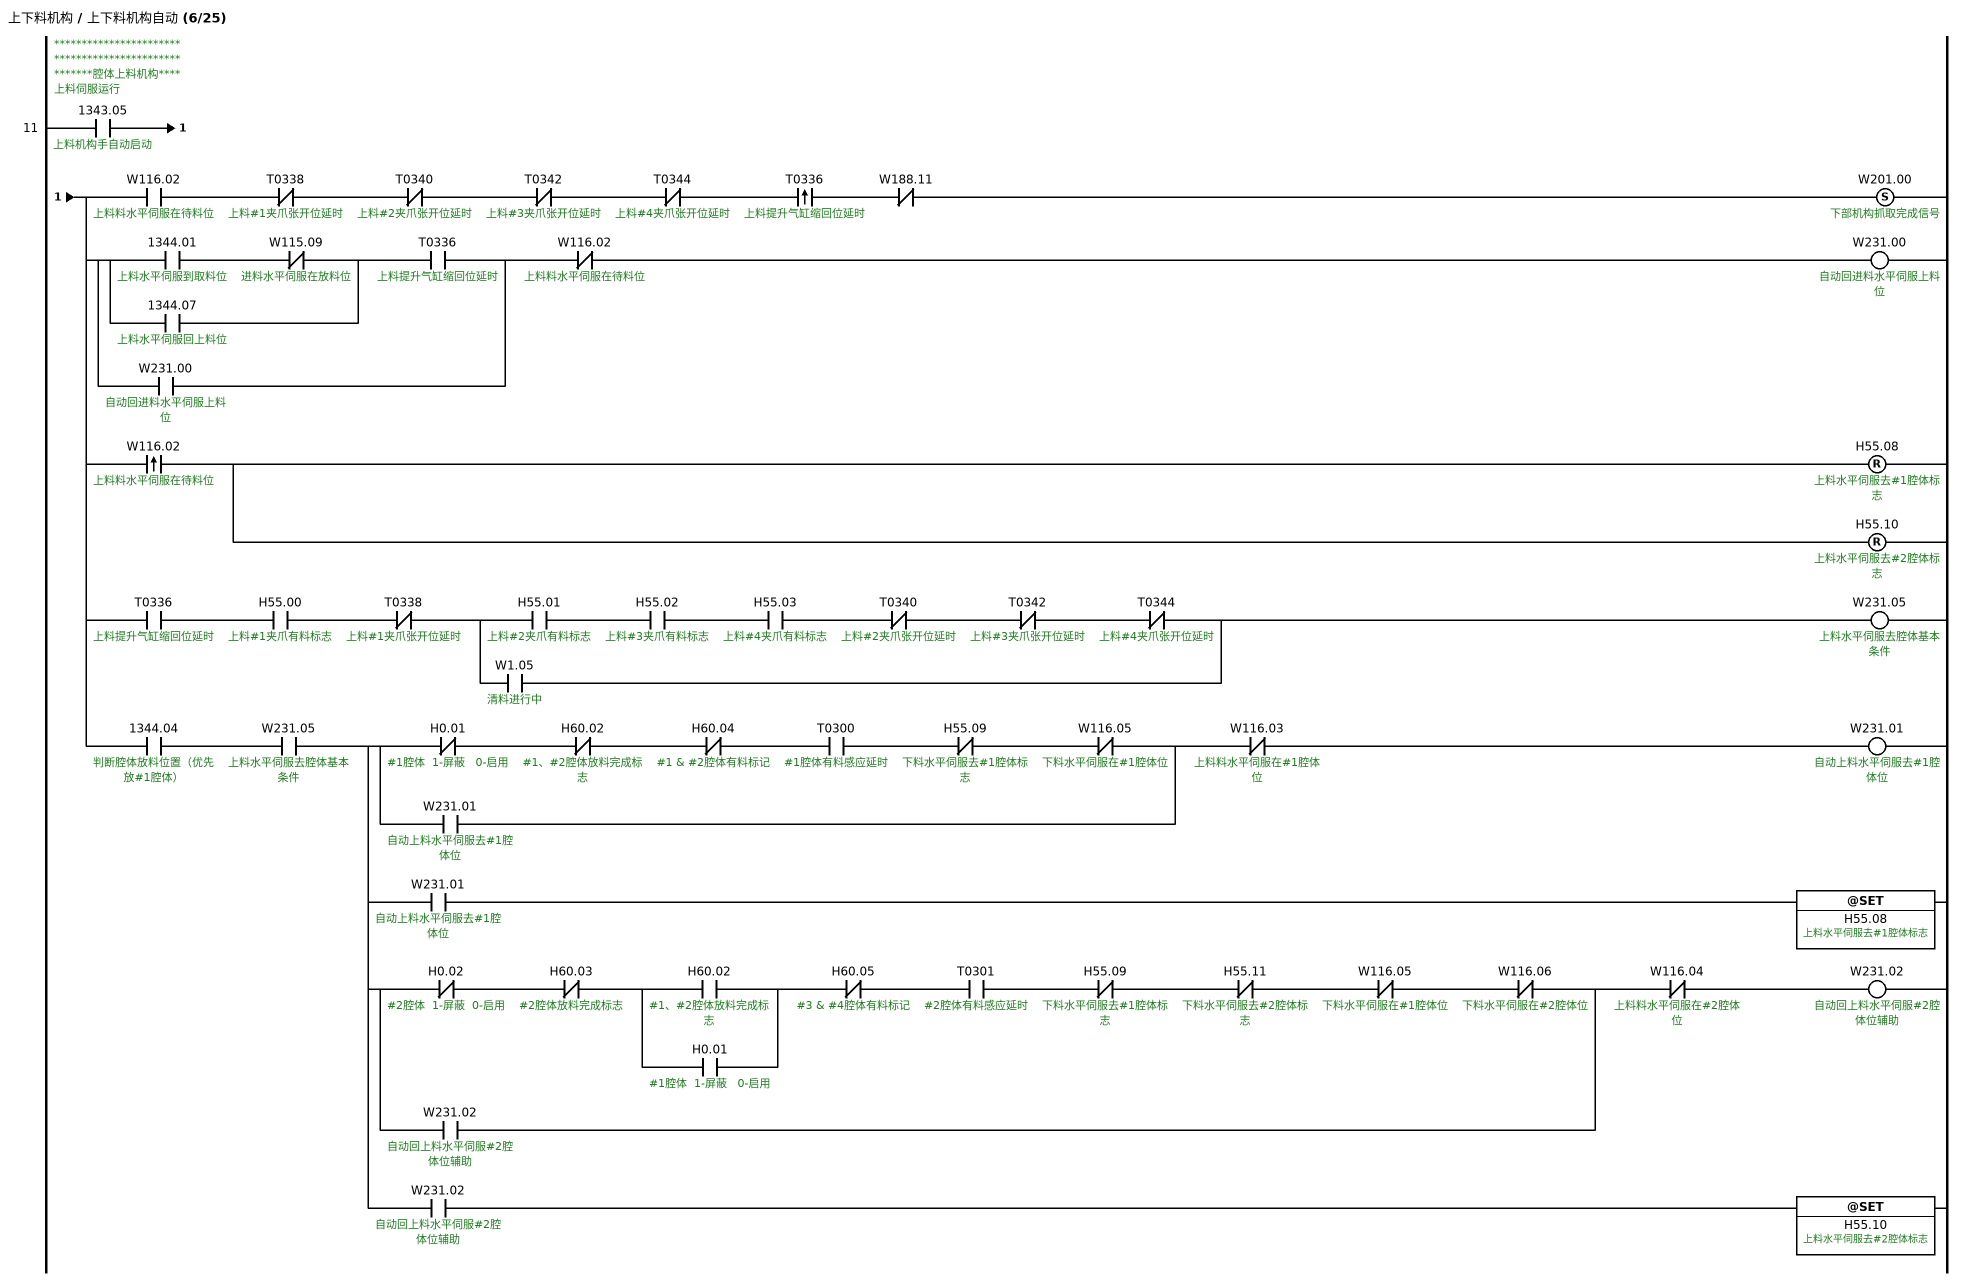
; rung 11: *********************** / *********************** / *******腔体上料机构**** / 上料伺服运行
LD 1343.05  ; 上料机构手自动启动
OUT TR0
AND W116.02  ; 上料料水平伺服在待料位
ANDNOT T0338  ; 上料#1夹爪张开位延时
ANDNOT T0340  ; 上料#2夹爪张开位延时
ANDNOT T0342  ; 上料#3夹爪张开位延时
ANDNOT T0344  ; 上料#4夹爪张开位延时
@AND T0336  ; 上料提升气缸缩回位延时
ANDNOT W188.11
SET W201.00  ; 下部机构抓取完成信号
LD TR0
LD 1344.01  ; 上料水平伺服到取料位
ANDNOT W115.09  ; 进料水平伺服在放料位
OR 1344.07  ; 上料水平伺服回上料位
AND T0336  ; 上料提升气缸缩回位延时
OR W231.00  ; 自动回进料水平伺服上料位
ANDLD
ANDNOT W116.02  ; 上料料水平伺服在待料位
OUT W231.00  ; 自动回进料水平伺服上料位
LD TR0
@AND W116.02  ; 上料料水平伺服在待料位
RSET H55.08  ; 上料水平伺服去#1腔体标志
RSET H55.10  ; 上料水平伺服去#2腔体标志
LD TR0
AND T0336  ; 上料提升气缸缩回位延时
AND H55.00  ; 上料#1夹爪有料标志
ANDNOT T0338  ; 上料#1夹爪张开位延时
LD H55.01  ; 上料#2夹爪有料标志
AND H55.02  ; 上料#3夹爪有料标志
AND H55.03  ; 上料#4夹爪有料标志
ANDNOT T0340  ; 上料#2夹爪张开位延时
ANDNOT T0342  ; 上料#3夹爪张开位延时
ANDNOT T0344  ; 上料#4夹爪张开位延时
OR W1.05  ; 清料进行中
ANDLD
OUT W231.05  ; 上料水平伺服去腔体基本条件
LD TR0
AND 1344.04  ; 判断腔体放料位置（优先放#1腔体）
AND W231.05  ; 上料水平伺服去腔体基本条件
OUT TR0
LDNOT H0.01  ; #1腔体  1-屏蔽   0-启用
ANDNOT H60.02  ; #1、#2腔体放料完成标志
ANDNOT H60.04  ; #1 & #2腔体有料标记
AND T0300  ; #1腔体有料感应延时
ANDNOT H55.09  ; 下料水平伺服去#1腔体标志
ANDNOT W116.05  ; 下料水平伺服在#1腔体位
OR W231.01  ; 自动上料水平伺服去#1腔体位
ANDLD
ANDNOT W116.03  ; 上料料水平伺服在#1腔体位
OUT W231.01  ; 自动上料水平伺服去#1腔体位
LD TR0
AND W231.01  ; 自动上料水平伺服去#1腔体位
@SET H55.08  ; 上料水平伺服去#1腔体标志
LD TR0
LDNOT H0.02  ; #2腔体  1-屏蔽  0-启用
ANDNOT H60.03  ; #2腔体放料完成标志
LD H60.02  ; #1、#2腔体放料完成标志
OR H0.01  ; #1腔体  1-屏蔽   0-启用
ANDLD
ANDNOT H60.05  ; #3 & #4腔体有料标记
AND T0301  ; #2腔体有料感应延时
ANDNOT H55.09  ; 下料水平伺服去#1腔体标志
ANDNOT H55.11  ; 下料水平伺服去#2腔体标志
ANDNOT W116.05  ; 下料水平伺服在#1腔体位
ANDNOT W116.06  ; 下料水平伺服在#2腔体位
OR W231.02  ; 自动回上料水平伺服#2腔体位辅助
ANDLD
ANDNOT W116.04  ; 上料料水平伺服在#2腔体位
OUT W231.02  ; 自动回上料水平伺服#2腔体位辅助
LD TR0
AND W231.02  ; 自动回上料水平伺服#2腔体位辅助
@SET H55.10  ; 上料水平伺服去#2腔体标志

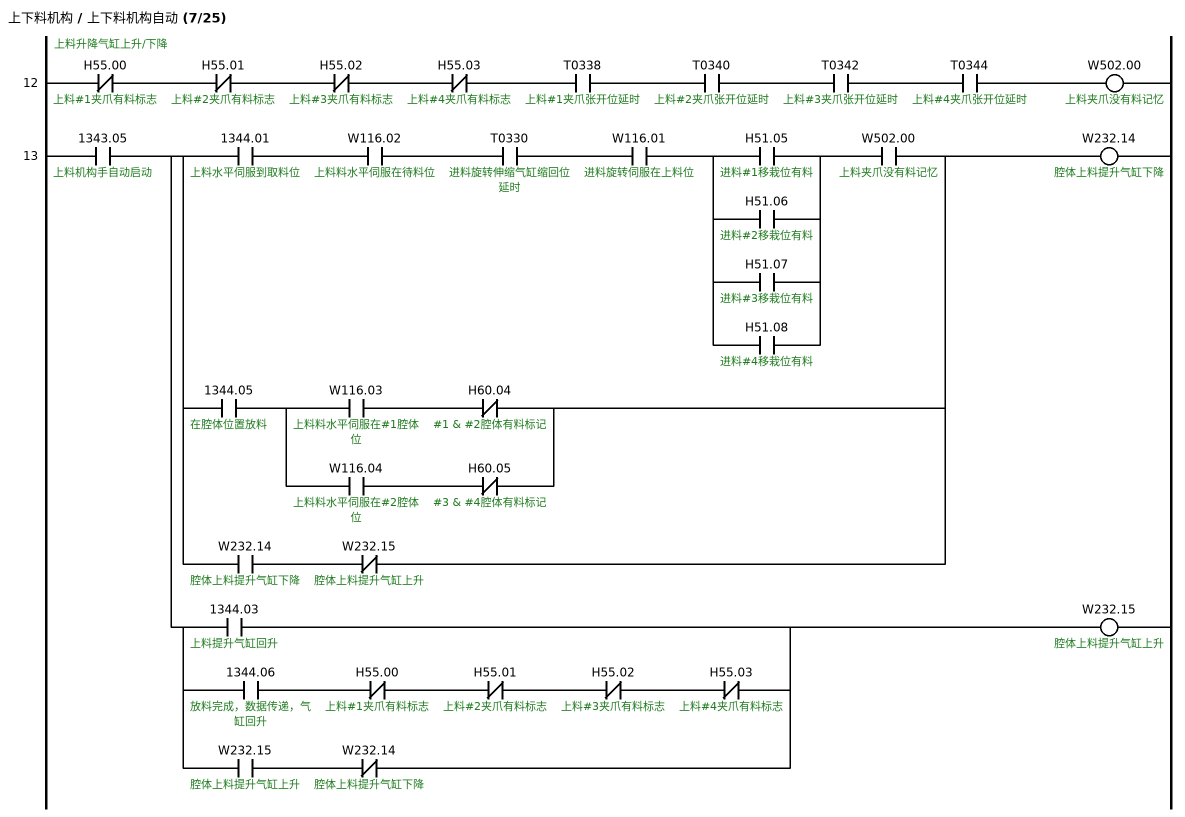
; rung 12: 上料升降气缸上升/下降
LDNOT H55.00  ; 上料#1夹爪有料标志
ANDNOT H55.01  ; 上料#2夹爪有料标志
ANDNOT H55.02  ; 上料#3夹爪有料标志
ANDNOT H55.03  ; 上料#4夹爪有料标志
AND T0338  ; 上料#1夹爪张开位延时
AND T0340  ; 上料#2夹爪张开位延时
AND T0342  ; 上料#3夹爪张开位延时
AND T0344  ; 上料#4夹爪张开位延时
OUT W502.00  ; 上料夹爪没有料记忆
; rung 13
LD 1343.05  ; 上料机构手自动启动
OUT TR0
LD 1344.01  ; 上料水平伺服到取料位
AND W116.02  ; 上料料水平伺服在待料位
AND T0330  ; 进料旋转伸缩气缸缩回位延时
AND W116.01  ; 进料旋转伺服在上料位
LD H51.05  ; 进料#1移栽位有料
OR H51.06  ; 进料#2移栽位有料
OR H51.07  ; 进料#3移栽位有料
OR H51.08  ; 进料#4移栽位有料
ANDLD
AND W502.00  ; 上料夹爪没有料记忆
LD 1344.05  ; 在腔体位置放料
LD W116.03  ; 上料料水平伺服在#1腔体位
ANDNOT H60.04  ; #1 & #2腔体有料标记
LD W116.04  ; 上料料水平伺服在#2腔体位
ANDNOT H60.05  ; #3 & #4腔体有料标记
ORLD
ANDLD
ORLD
LD W232.14  ; 腔体上料提升气缸下降
ANDNOT W232.15  ; 腔体上料提升气缸上升
ORLD
ANDLD
OUT W232.14  ; 腔体上料提升气缸下降
LD TR0
LD 1344.03  ; 上料提升气缸回升
LD 1344.06  ; 放料完成，数据传递，气缸回升
ANDNOT H55.00  ; 上料#1夹爪有料标志
ANDNOT H55.01  ; 上料#2夹爪有料标志
ANDNOT H55.02  ; 上料#3夹爪有料标志
ANDNOT H55.03  ; 上料#4夹爪有料标志
ORLD
LD W232.15  ; 腔体上料提升气缸上升
ANDNOT W232.14  ; 腔体上料提升气缸下降
ORLD
ANDLD
OUT W232.15  ; 腔体上料提升气缸上升

